{attribute 'GeneratedUsingTerminal: AT2050-0500-0018'}
{attribute addProperty BoxType "AT2050-0500-0018"}
{attribute addProperty Id "A_0095_AT2021_5250_0019_AT2021_5250AT2021_33A3DF1B80"}
{attribute addProperty CRC "3420870056"}
{attribute addProperty Size "80"}
TYPE A_0049_AT2050_0500_0018_CBE655A8 EXTENDS AT2050_2EA6C9BF :
STRUCT
	{attribute addProperty Name "A_0095_AT2021_5250_0019_AT2021_5250"}
	{attribute addProperty PreviousPort "A_0049(AT2050-0500-0018) : B"}
	A_0095_AT2021_5250_0019_AT2021_5250 : AT2021_33A3DF1B;
END_STRUCT
END_TYPE

(* stored: Version 1.2.0.0, ProductVersion 3.1.4024.9
   DUT A_0049_AT2050_0500_0018_CBE655A8: Id {4a09bcdd-5d71-4a7d-964d-d024e78a07c8} *)
